FUNCTION_BLOCK FB_Scale
VAR_INPUT
END_VAR
VAR_OUTPUT
END_VAR
VAR
END_VAR

END_FUNCTION_BLOCK

(* stored: Version 1.1.0.1
   POU FB_Scale: Id {5d67843b-3530-4c9b-9c4d-73d68b9ee1cc}, SpecialFunc None *)
